FUNCTION_BLOCK FB_boundaryForceFeedback
VAR_INPUT
END_VAR
VAR_OUTPUT
END_VAR

VAR
	// force control parameters in local tip coordinate
//	m_oriKp :Vec3d :=[1, 1, 0.5];
//	m_oriKd :Vec3d :=[0.04,0.04, 0.01];
	m_oriKp :Vec3d :=[0.2, 0.2, 0.1];
	m_oriKd :Vec3d :=[0.02,0.02, 0.005];

	m_oriCartTrq,m_oriCartTrqLocal :Vec3d;
	
	m_posKp :LREAL := 200;
	m_posKd :LREAL := 10;
	m_posCartForce:Vec3d;
	
	
END_VAR

METHOD run : Vec7d

VAR_IN_OUT CONSTANT
	i_slaveIdx :INT;
	i_shoulderPose :ST_Frame;
	i_masterArm :FB_MasterArm;
	i_slaveStatus :ST_SlaveStatus;
END_VAR

VAR
	posErrInScope, oriErrInScope:Vec3d;
	posErr, oriErr:Vec3d;
	posErrLocal, oriErrLocal :Vec3d;
	vel, velLocal, wVel,wVelLocal :Vec3d;
	oriErrAxis, wVelProj :Vec3d;
	rotInv :Mat3d;
	oriJaco, oriJacoT :Mat3d;
	oriJntTrq :Vec3d;
	
	i,j:INT;
	posErrAxis, velProj :Vec3d;
	posJaco, posJacoT :Mat3d;
	posJntTrq :Vec3d;
	
	trqScale :LREAL;
END_VAR
run:=g_zeroVec7d;

FOR i:=1 TO 3 DO
	posErrInScope[i]:= -i_slaveStatus.m_masterSlavePoseError[i_slaveIdx][i];
	oriErrInScope[i]:= -i_slaveStatus.m_masterSlavePoseError[i_slaveIdx][i+3];
	vel[i]:=i_masterArm.curCartTwist[i];
	wVel[i]:=i_masterArm.curCartTwist[i+3];
END_FOR

// calculate pose error in shoulder coordinate
matTranspose(i_shoulderPose.m_rot, rotInv);
matMultiVec(rotInv, posErrInScope, posErr);
matMultiVec(rotInv, oriErrInScope, oriErr);
// ################### 	force  #########################
// add threshold
IF norm(posErr) > g_smallNum THEN
	// project error in tip coordinate
	matTranspose(i_masterArm.curCartPose.m_rot, rotInv);
	matMultiVec(rotInv, posErr, posErrLocal);
	matMultiVec(rotInv, oriErr, oriErrLocal);
	matMultiVec(rotInv, vel, velLocal);
	matMultiVec(rotInv, wVel, wVelLocal);
	
	// compute velocity in error direction
	posErrAxis := posErr;
	normalize(posErrAxis);
	vecMultiNum(posErrAxis, vecDot(vel, posErrAxis), velProj);
	
	// compute local cartesion torque
	FOR i:=1 TO 3 DO
		m_posCartForce[i]:= m_posKp * posErr[i]-m_posKd*velProj[i];
	END_FOR
	
	// compute joint space torque
	FOR i :=1 TO  3 DO
		FOR j:=1 TO 3 DO
			posJaco[i,j]:= i_masterArm.jaco[i,j];
		END_FOR
	END_FOR
	matTranspose(posJaco, posJacoT);
	matMultiVec(posJacoT, m_posCartForce, posJntTrq);
	
	// scale joint troque
	trqScale := 1;
	FOR i:=1 TO 3 DO 
		trqScale:=MAX(trqScale, ABS(posJntTrq[i]/GVL_ArmJointParameters.g_jntMaxTrq[i]));
	END_FOR
	
	run[1]:=posJntTrq[1]/trqScale;
	run[2]:=posJntTrq[2]/trqScale;
	run[3]:=posJntTrq[3]/trqScale;
END_IF


// ###################  torque #########################
// add threshold
IF norm(oriErr) > g_smallNum THEN
	// project error in tip coordinate
	matTranspose(i_masterArm.curCartPose.m_rot, rotInv);
	matMultiVec(rotInv, posErr, posErrLocal);
	matMultiVec(rotInv, oriErr, oriErrLocal);
	matMultiVec(rotInv, vel, velLocal);
	matMultiVec(rotInv, wVel, wVelLocal);
	
	// compute velocity in error direction
	oriErrAxis := oriErrLocal;
	normalize(oriErrAxis);
	vecMultiNum(oriErrAxis, vecDot(wVelLocal, oriErrAxis), wVelProj);
	
	// compute local cartesion torque
	FOR i:=1 TO 3 DO
		m_oriCartTrqLocal[i]:= m_oriKp[i] * oriErrLocal[i]-m_oriKd[i]*wVelProj[i];
	END_FOR
	
	// project torque back to shoulder coordinate
	matMultiVec(i_masterArm.curCartPose.m_rot, m_oriCartTrqLocal, m_oriCartTrq);
	
	// compute joint space torque
	// for simplicity, we current only use last 3 joint for torque feedback
	FOR i :=1 TO  3 DO
		FOR j:=1 TO 3 DO
			oriJaco[i,j]:= i_masterArm.jaco[i+3,j+4];
		END_FOR
	END_FOR
	matTranspose(oriJaco, oriJacoT);
	matMultiVec(oriJacoT, m_oriCartTrq, oriJntTrq);
	
	// scale joint troque
	trqScale := 1;
	FOR i:=1 TO 3 DO 
		trqScale:=MAX(trqScale, ABS(oriJntTrq[i]/GVL_ArmJointParameters.g_jntMaxTrq[i+4]));
	END_FOR
	
	run[5]:=oriJntTrq[1]/trqScale;
	run[6]:=oriJntTrq[2]/trqScale;
	run[7]:=oriJntTrq[3]/trqScale;
END_IF
END_METHOD

END_FUNCTION_BLOCK

(* stored: Version 1.1.0.1, ProductVersion 3.1.4024.12
   POU FB_boundaryForceFeedback: Id {0a761a35-a81f-4506-87e3-40d8a9b51e60}, SpecialFunc None
   Method run: Id {85672461-4205-4eb7-9251-08e742de258a} *)
